(* CODESYS project DeanPowerSupplyComponent (1).library
   Author: Lily Dollard, Scott Kinder
   Version: 2025.10.20.11
   Title: Nemo
   Placeholder: Nemo
   Company: Photara

Project tree, tasks and I/O mapping:
  libraries: Base, 2025.10.13.11 (Photara); Tc2_Math, * (Beckhoff Automation GmbH); Tc2_Standard, * (Beckhoff Automation GmbH); Tc2_System, * (Beckhoff Automation GmbH); Tc2_Utilities, * (Beckhoff Automation GmbH)
  DUTs/
    data type ST_PowerSupplyCalibration
    data type ST_PowerSupplyConfiguration
    data type ST_PowerSupplyStatus
  GVLs/
    global variables GC_Dean
    global variables GPL_Dean
  ITFs/
    interface I_PowerSupply: Disable_HV, Enable_HV, InjectConfiguration, P_PowerSupplyStatus
    interface I_PowerSupplyConfiguration: P_PowerSupplyConfiguration
    interface I_PowerSupplyExt: GetCurrent, GetVoltage, InputPowerOff, InputPowerOn, SetCurrent, SetVoltage
    interface I_PowerSupplySystem: ClearErrors, Disable_HV, Enable_HV, FullShutDown, InputPowerOff, InputPowerOn, SetCurrent, SetVoltage
  POUs/
    function block FB_DeanPowerSupply [ST]: _DeanCyclic, _InitializeReferences, _SetCommandPermIntlkConfiguration, _UpdateComponentStatus, _ComponentCyclic, _EvaluateCompletionConditions, CyclicLogic, Disable_HV, Enable_HV, GetCurrent, GetVoltage, InputPowerOff, InputPowerOn, SetCurrent, SetVoltage, Check_Results, Test_Disable_HV, Test_Enable_HV, Test_GetCurrent, Test_GetVoltage, Test_InputPowerOff, Test_InputPowerOn, Test_SetCurrent, Test_SetVoltage, CheckForErrors, ClearErrors, InjectConfiguration, Interpolate, P_PowerSupplyConfiguration, P_PowerSupplyStatus
    function block FB_HVPS_System [ST]: _Initialize, _InitializeChildrenDependencies, _SetDependencyConfiguration, CyclicLogic, FB_Init, P_supply_status, RunTests, ClearErrors, Disable_HV, Enable_HV, FullShutDown, InputPowerOff, InputPowerOn, SetCurrent, SetVoltage
    program MAIN [ST]
  VISUs/
*)

// DUTs/ST_PowerSupplyCalibration
TYPE ST_PowerSupplyCalibration :
STRUCT
	VSET_Scale		: LREAL 	:= 1.000;
	VSET_Offset		: LREAL  := 0; // V
	ISET_Scale		: LREAL	:= 1.000;
	ISET_Offset		: LREAL  := 0; // mA
	                  
	VMON_Scale		: LREAL 	:= 1.000;
	VMON_Offset		: LREAL  := 0; // V
	IMON_Scale		: LREAL 	:= 1.000;
	IMON_Offset		: LREAL  := 0; // mA
END_STRUCT
END_TYPE

// DUTs/ST_PowerSupplyConfiguration
TYPE ST_PowerSupplyConfiguration :
STRUCT
	ComponentConfiguration : REFERENCE TO Base.ST_ComponentConfiguration;
	
	// Supply Characteristics
	IsPositive		: BOOL; 			// Sends negative monitor values to the HMI if False
	
	MinVoltage 		: LREAL := 0; 		// Minimum voltage (V) that the user can specify, usually 0
	MaxVoltageAbs 	: LREAL;			// Maximum voltage (V) that the user can specify
	MinCurrent		: LREAL := 0;		// Minimum current (mA) that the user can specify, usually 0
	MaxCurrent		: LREAL;			// Maximum current (mA) that the user can specify
	
	HasVMON			: BOOL 	:= TRUE; 	// Can the user watch the voltage output?
	HasIMON			: BOOL 	:= TRUE; 	// Can the user watch the current output?
	HasVSET			: BOOL 	:= TRUE;	// Can the user specify a desired voltage?
	HasISET			: BOOL 	:= TRUE; 	// Can the user specify maximum current?
	
	NeedsVREF		: BOOL ; 			// False if the reference voltage for control inputs is generated internally
	VREF			: LREAL;			// Reference voltage for control inputs
	plc_VREF		: INT;
	
	VSET_needs_ramp	: BOOL 	:= FALSE;	// False allows the full V value to be set immediately
	Ramp_increment	: LREAL := 10.0;   	// Voltage (V) to step up at a time after checking that current is within acceptable limits
	
	// Control signal characteristics
	plc_min_IMON  	: INT 	:= 0;    	// PLC signal corresponding to the minimum current reading
	plc_max_IMON  	: INT 	:= 32767; 	// PLC signal corresponding to the maximum current reading
	                                                                      
	plc_min_ISET  	: INT 	:= 0;	  	// PLC signal corresponding to the minimum current setting
	plc_max_ISET  	: INT 	:= 32767; 	// PLC signal corresponding to the maximum current setting
	
	plc_min_VMON  	: INT 	:= 0;     	// PLC signal corresponding to the minimum voltage reading
	plc_max_VMON  	: INT 	:= 32767;	// PLC signal corresponding to the maximum voltage reading
	                                                                         
	plc_min_VSET  	: INT 	:= 0;	  	// PLC signal corresponding to the minimum voltage setting
	plc_max_VSET  	: INT 	:= 32767; 	// PLC signal corresponding to the maximum voltage setting
	
	// Error Conditions
	OverCurrentErrorThreshold 		: LREAL := 1.05;	// over-current level, relative to IMON, to disable the output
	OverVoltageErrorThreshold 		: LREAL := 1.05;	// over-voltage level, relative to VSET, to disable the output
	MaxVoltageBuffer				: LREAL := 100.0;	// volts beyond MaxVoltageAbs to allow before killing supply power
	UnderVoltageWarningThreshold 	: LREAL := 0.95;	// under-voltage level, relative to VSET, to warn setpoint is not met
	
	ClearErrors : BOOL := FALSE;
	
	// Calibration
	Calibration		: ST_PowerSupplyCalibration;
	
	// Setpoints
	VSET			: LREAL;	// V
	ISET			: LREAL;	// mA
	POWERED			: BOOL;	
	ENABLED			: BOOL;
	
END_STRUCT
END_TYPE

// DUTs/ST_PowerSupplyStatus
TYPE ST_PowerSupplyStatus :
STRUCT
	BaseComponentStatus : REFERENCE TO Base.ST_ComponentStatus;
	
	// Controls mapped to PLC terminals
	VSET_to_plc 		AT %Q* : INT;
	ISET_to_plc 		AT %Q* : INT;
	VREF_to_plc			AT %Q* : INT;
	VMON_from_plc 		AT %I* : INT;
	IMON_from_plc 		AT %I* : INT;
	POWERED				AT %Q* : BOOL; 
	ENABLED				AT %Q* : BOOL;
	
	// Live outputs of the HV supply, translated into real units
	VMON 		: LREAL;	// V
	IMON		: LREAL;	// mA
	
	// Most recent settings given to the power supply
	VSET		: LREAL;
	ISET		: LREAL;
	
	V_was_set 	: BOOL; // flag for successful voltage set
	
	UnderVoltageWarning			: BOOL := FALSE;
	CurrentLimitWarning			: BOOL := FALSE;
	
	OverVoltageSetpointError	: BOOL := FALSE;
	OverMaxVoltageError			: BOOL := FALSE;
	
	OverCurrentSetpointError	: BOOL := FALSE;
	OverMaxCurrentError			: BOOL := FALSE;
	
	ErrorsAreClear					: BOOL := TRUE;
	
END_STRUCT
END_TYPE

// GVLs/GC_Dean
{attribute 'qualified_only'}
{attribute 'global_init_slot' := '41600'}
VAR_GLOBAL CONSTANT
	INDEX_COMMAND_MIN : DINT := GPL_Dean.INDEX_COMMAND_MIN;  
	INDEX_COMMAND_MAX : DINT := GPL_Dean.INDEX_COMMAND_MAX;
END_VAR

// GVLs/GPL_Dean
{attribute 'qualified_only'}
{attribute 'global_init_slot' := '41500'}
VAR_GLOBAL CONSTANT
	INDEX_COMMAND_MIN : DINT := 0;  
	INDEX_COMMAND_MAX : DINT := 5;
END_VAR

// ITFs/I_PowerSupply
// Basic high-voltage power supply that can turn on or off
INTERFACE I_PowerSupply EXTENDS I_BaseCyclic

// Shut off the output voltage
METHOD Disable_HV
VAR_INPUT
END_VAR
END_METHOD

// Turn on the output voltage
METHOD Enable_HV
VAR_INPUT
END_VAR
END_METHOD

METHOD InjectConfiguration
VAR_INPUT
	PowerSupplyConfiguration : REFERENCE TO ST_PowerSupplyConfiguration;
END_VAR
END_METHOD

PROPERTY P_PowerSupplyStatus : REFERENCE TO ST_PowerSupplyStatus
GET
END_GET
END_PROPERTY

END_INTERFACE

// ITFs/I_PowerSupplyConfiguration
// Basic high-voltage power supply that can turn on or off
INTERFACE I_PowerSupplyConfiguration EXTENDS __SYSTEM.IQueryInterface

PROPERTY P_PowerSupplyConfiguration : REFERENCE TO ST_PowerSupplyConfiguration
GET
END_GET
END_PROPERTY

END_INTERFACE

// ITFs/I_PowerSupplyExt
(*
Additional power supply capabilities:
* Adds a distinction between input power and the existing controls for HV output enable/disable
* Allows setting a desired output voltage and current
* Monitors the actual voltage and current
*)

INTERFACE I_PowerSupplyExt EXTENDS I_PowerSupply

// Read the currently-output current in milliamps (mA)
METHOD GetCurrent
END_METHOD

// Read the currently-output voltage in Volts (V)
METHOD GetVoltage
END_METHOD

// Turn off power to the supply
METHOD InputPowerOff
END_METHOD

// Turn on power to the supply
METHOD InputPowerOn
END_METHOD

// Send the the desired or maximum current setpoint (in mA) to the power supply
METHOD SetCurrent
VAR_INPUT
	setpoint : LREAL; // mA
END_VAR
END_METHOD

// Send the the voltage setpoint (V) to the power supply
METHOD SetVoltage
VAR_INPUT
	setpoint : LREAL; // V
END_VAR
END_METHOD

END_INTERFACE

// ITFs/I_PowerSupplySystem
INTERFACE I_PowerSupplySystem EXTENDS __SYSTEM.IQueryInterface

METHOD ClearErrors : BOOL
VAR_INPUT
	Index : DINT;
END_VAR
END_METHOD

(* Shut off the output voltage*)
METHOD Disable_HV
VAR_INPUT
	Index : DINT;
END_VAR
END_METHOD

{warning 'Add method implementation '}
(* Turn on the output voltage*)
METHOD Enable_HV
VAR_INPUT
	Index : DINT;
END_VAR
END_METHOD

METHOD FullShutDown : BOOL
VAR_INPUT
END_VAR
END_METHOD

{warning 'Add method implementation '}
(* Turn off power to the supply*)
METHOD InputPowerOff
VAR_INPUT
	Index : DINT;
END_VAR
END_METHOD

{warning 'Add method implementation '}
(* Turn on power to the supply*)
METHOD InputPowerOn
VAR_INPUT
	Index : DINT;
END_VAR
END_METHOD

{warning 'Add method implementation '}
(* Send the the desired or maximum current setpoint (in mA) to the power supply*)
METHOD SetCurrent
VAR_INPUT
	(* mA*)
	setpoint	: LREAL;
	Index : DINT;
END_VAR
END_METHOD

{warning 'Add method implementation '}
(* Send the the voltage setpoint (V) to the power supply*)
METHOD SetVoltage
VAR_INPUT
	(* V*)
	setpoint	: LREAL;
	Index : DINT;
END_VAR
END_METHOD

END_INTERFACE

// POUs/FB_DeanPowerSupply
FUNCTION_BLOCK FB_DeanPowerSupply EXTENDS Base.FB_Component<GC_Dean.INDEX_COMMAND_MIN,GC_Dean.INDEX_COMMAND_MAX> IMPLEMENTS I_PowerSupplyExt, I_PowerSupplyConfiguration
VAR CONSTANT
	INDEX_COMMAND_Enable_HV 		: INT := 0;
	INDEX_COMMAND_Disable_HV 		: INT := 1;
	INDEX_COMMAND_InputPowerOn		: INT := 2;
	INDEX_COMMAND_InputPowerOff 	: INT := 3;
	INDEX_COMMAND_SetVoltage 		: INT := 4;
	INDEX_COMMAND_SetCurrent		: INT := 5;
	
END_VAR

VAR
//	ComponentConfiguration : Base.ST_ComponentConfiguration;
	
//	_iInjectedConfiguration		: I_PowerSupplyConfiguration;
	
	Run_Tests_Trigger : BOOL := FALSE;
END_VAR

VAR_INPUT
	DeanConfig 		: ST_PowerSupplyConfiguration;
	DeanStatus		: ST_PowerSupplyStatus;
END_VAR

METHOD PROTECTED _DeanCyclic
VAR_INST
// 	VSET_actual	: LREAL;
// 	ISET_actual : LREAL;
END_VAR
// Reset errors if requested
IF DeanConfig.ClearErrors THEN
	ClearErrors();
	DeanConfig.ClearErrors := FALSE;
END_IF

// Turn on or off power if the config requests it
IF DeanStatus.POWERED <> DeanConfig.POWERED THEN
	IF DeanConfig.POWERED THEN
		InputPowerOn();
	ELSE
		InputPowerOff();
		DeanConfig.ENABLED := FALSE;
	END_IF
END_IF

// Enable or disable HV if the config requests it
IF DeanStatus.ENABLED <> DeanConfig.ENABLED THEN
	IF DeanConfig.ENABLED AND DeanConfig.POWERED THEN
		Enable_HV();
	ELSE
		DeanConfig.ENABLED := FALSE;
		Disable_HV();
	END_IF
END_IF

// get the actual last settings sent to the PLC (Config values are nominal)
// VSET_actual		:= DeanConfig.VSET * DeanConfig.Calibration.VSET_Scale + DeanConfig.Calibration.VSET_Offset;
// VSET_actual 	:= MAX(DeanConfig.MinVoltage, VSET_actual);
// VSET_actual 	:= MIN(VSET_actual, DeanConfig.MaxVoltageAbs);
// 
// ISET_actual		:= DeanConfig.ISET * DeanConfig.Calibration.ISET_Scale + DeanConfig.Calibration.ISET_Offset;
// ISET_actual 	:= MAX(DeanConfig.MinCurrent, ISET_actual);
// ISET_actual 	:= MIN(ISET_actual, DeanConfig.MaxCurrent);

// Send the desired values to the PLC if the input has changed
IF DeanConfig.HasVSET THEN
	// IF VSET_actual <> DeanStatus.VSET AND NOT (SUPER^.Commands[INDEX_COMMAND_SetVoltage].Busy) THEN
		SetVoltage(DeanConfig.VSET);
	// END_IF
END_IF

IF DeanConfig.HasISET THEN
	// IF ISET_actual <> DeanStatus.ISET THEN
		SetCurrent(DeanConfig.ISET);
	// END_IF
END_IF

// Monitor for errors (monitor pins only work when powered on)
IF DeanStatus.POWERED THEN
	CheckForErrors();
END_IF
END_METHOD

METHOD PROTECTED _InitializeReferences : BOOL
//Initialize data references
BaseConfiguration.InstancePath 						REF= InstancePath;

ComponentConfiguration.BaseConfiguration 			REF= SUPER^.BaseConfiguration;
                                                    
ComponentStatus.BaseStatus							REF= SUPER^.BaseStatus;

ComponentStatus.AmsNetId							REF= ComponentConfiguration.AmsNetId;

DeanConfig.ComponentConfiguration					REF= SUPER^.ComponentConfiguration;

DeanStatus.BaseComponentStatus						REF= SUPER^.ComponentStatus;

_InitializeReferences 								:= TRUE; // apply at end of all reference initialization
END_METHOD

METHOD PROTECTED _SetCommandPermIntlkConfiguration : BOOL
//Enable HV
CommandPermIntlkConfiguration[INDEX_COMMAND_Enable_HV].P_CommandConfiguration.CommandDescription := 'Enable Power Supply Output';
CommandPermIntlkConfiguration[INDEX_COMMAND_Enable_HV].P_CommandConfiguration.CommandIndex := INDEX_COMMAND_Enable_HV;
CommandPermIntlkConfiguration[INDEX_COMMAND_Enable_HV].P_CommandConfiguration.CommandPOUName := 'Enable_HV';
CommandPermIntlkConfiguration[INDEX_COMMAND_Enable_HV].P_CommandConfiguration.Priority := Base.E_CommandPriority.Priority_Normal;
CommandPermIntlkConfiguration[INDEX_COMMAND_Enable_HV].P_CommandConfiguration.TimeoutTime := T#200MS;
CommandPermIntlkConfiguration[INDEX_COMMAND_Enable_HV].P_CommandConfiguration.CompletionCondition REF= SUPER^.CommandCompletionConditions[INDEX_COMMAND_Enable_HV];

CommandPermIntlkConfiguration[INDEX_COMMAND_Enable_HV].P_PermIntlkConfiguration.PermIntlkObj[0].Condition REF= DeanStatus.POWERED;
CommandPermIntlkConfiguration[INDEX_COMMAND_Enable_HV].P_PermIntlkConfiguration.PermIntlkObj[0].Description := 'Powered on';
CommandPermIntlkConfiguration[INDEX_COMMAND_Enable_HV].P_PermIntlkConfiguration.PermIntlkObj[0].Index := 0;

CommandPermIntlkConfiguration[INDEX_COMMAND_Enable_HV].P_PermIntlkConfiguration.PermIntlkObj[1].Condition REF= DeanStatus.ErrorsAreClear;
CommandPermIntlkConfiguration[INDEX_COMMAND_Enable_HV].P_PermIntlkConfiguration.PermIntlkObj[1].Description := 'No voltage or current errors';
CommandPermIntlkConfiguration[INDEX_COMMAND_Enable_HV].P_PermIntlkConfiguration.PermIntlkObj[1].Index := 1;

//Disable HV
CommandPermIntlkConfiguration[INDEX_COMMAND_Disable_HV].P_CommandConfiguration.CommandDescription := 'Disable Power Supply Output';
CommandPermIntlkConfiguration[INDEX_COMMAND_Disable_HV].P_CommandConfiguration.CommandIndex := INDEX_COMMAND_Disable_HV;
CommandPermIntlkConfiguration[INDEX_COMMAND_Disable_HV].P_CommandConfiguration.CommandPOUName := 'Disable_HV';
CommandPermIntlkConfiguration[INDEX_COMMAND_Disable_HV].P_CommandConfiguration.Priority := Base.E_CommandPriority.Priority_High;
CommandPermIntlkConfiguration[INDEX_COMMAND_Disable_HV].P_CommandConfiguration.TimeoutTime := T#200MS;
CommandPermIntlkConfiguration[INDEX_COMMAND_Disable_HV].P_CommandConfiguration.CompletionCondition REF= SUPER^.CommandCompletionConditions[INDEX_COMMAND_Disable_HV];

//Input power on
CommandPermIntlkConfiguration[INDEX_COMMAND_InputPowerOn].P_CommandConfiguration.CommandDescription := 'Provide input power to supply';
CommandPermIntlkConfiguration[INDEX_COMMAND_InputPowerOn].P_CommandConfiguration.CommandIndex := INDEX_COMMAND_InputPowerOn;
CommandPermIntlkConfiguration[INDEX_COMMAND_InputPowerOn].P_CommandConfiguration.CommandPOUName := 'InputPowerOn';
CommandPermIntlkConfiguration[INDEX_COMMAND_InputPowerOn].P_CommandConfiguration.Priority := Base.E_CommandPriority.Priority_Normal;
CommandPermIntlkConfiguration[INDEX_COMMAND_InputPowerOn].P_CommandConfiguration.TimeoutTime := T#200MS;
CommandPermIntlkConfiguration[INDEX_COMMAND_InputPowerOn].P_CommandConfiguration.CompletionCondition REF= SUPER^.CommandCompletionConditions[INDEX_COMMAND_InputPowerOn];

CommandPermIntlkConfiguration[INDEX_COMMAND_InputPowerOn].P_PermIntlkConfiguration.PermIntlkObj[0].Condition REF= DeanStatus.ErrorsAreClear;
CommandPermIntlkConfiguration[INDEX_COMMAND_InputPowerOn].P_PermIntlkConfiguration.PermIntlkObj[0].Description := 'No voltage or current errors';
CommandPermIntlkConfiguration[INDEX_COMMAND_InputPowerOn].P_PermIntlkConfiguration.PermIntlkObj[0].Index := 0;

//Input power off
CommandPermIntlkConfiguration[INDEX_COMMAND_InputPowerOff].P_CommandConfiguration.CommandDescription := 'Cut off input power to supply';
CommandPermIntlkConfiguration[INDEX_COMMAND_InputPowerOff].P_CommandConfiguration.CommandIndex := INDEX_COMMAND_InputPowerOff;
CommandPermIntlkConfiguration[INDEX_COMMAND_InputPowerOff].P_CommandConfiguration.CommandPOUName := 'InputPowerOff';
CommandPermIntlkConfiguration[INDEX_COMMAND_InputPowerOff].P_CommandConfiguration.Priority := Base.E_CommandPriority.Priority_High;
CommandPermIntlkConfiguration[INDEX_COMMAND_InputPowerOff].P_CommandConfiguration.TimeoutTime := T#200MS;
CommandPermIntlkConfiguration[INDEX_COMMAND_InputPowerOff].P_CommandConfiguration.CompletionCondition REF= SUPER^.CommandCompletionConditions[INDEX_COMMAND_InputPowerOff];

//Set Voltage
CommandPermIntlkConfiguration[INDEX_COMMAND_SetVoltage].P_CommandConfiguration.CommandDescription := 'Set the desired HV output voltage';
CommandPermIntlkConfiguration[INDEX_COMMAND_SetVoltage].P_CommandConfiguration.CommandIndex := INDEX_COMMAND_SetVoltage;
CommandPermIntlkConfiguration[INDEX_COMMAND_SetVoltage].P_CommandConfiguration.CommandPOUName := 'SetVoltage';
CommandPermIntlkConfiguration[INDEX_COMMAND_SetVoltage].P_CommandConfiguration.Priority := Base.E_CommandPriority.Priority_Normal;
CommandPermIntlkConfiguration[INDEX_COMMAND_SetVoltage].P_CommandConfiguration.TimeoutTime := T#200MS;
CommandPermIntlkConfiguration[INDEX_COMMAND_SetVoltage].P_CommandConfiguration.CompletionCondition REF= SUPER^.CommandCompletionConditions[INDEX_COMMAND_SetVoltage];

CommandPermIntlkConfiguration[INDEX_COMMAND_SetVoltage].P_PermIntlkConfiguration.PermIntlkObj[0].Condition REF= DeanConfig.HasVSET;
CommandPermIntlkConfiguration[INDEX_COMMAND_SetVoltage].P_PermIntlkConfiguration.PermIntlkObj[0].Description := 'HVPS has VSET capability';
CommandPermIntlkConfiguration[INDEX_COMMAND_SetVoltage].P_PermIntlkConfiguration.PermIntlkObj[0].Index := 0;

CommandPermIntlkConfiguration[INDEX_COMMAND_SetVoltage].P_PermIntlkConfiguration.PermIntlkObj[1].Condition REF= DeanStatus.POWERED;
CommandPermIntlkConfiguration[INDEX_COMMAND_SetVoltage].P_PermIntlkConfiguration.PermIntlkObj[1].Description := 'Supply power is on, can set voltage';
CommandPermIntlkConfiguration[INDEX_COMMAND_SetVoltage].P_PermIntlkConfiguration.PermIntlkObj[1].Index := 1;

//Set Current
CommandPermIntlkConfiguration[INDEX_COMMAND_SetCurrent].P_CommandConfiguration.CommandDescription := 'Set the maximum current output from the HV terminals';
CommandPermIntlkConfiguration[INDEX_COMMAND_SetCurrent].P_CommandConfiguration.CommandIndex := INDEX_COMMAND_SetCurrent;
CommandPermIntlkConfiguration[INDEX_COMMAND_SetCurrent].P_CommandConfiguration.CommandPOUName := 'SetCurrent';
CommandPermIntlkConfiguration[INDEX_COMMAND_SetCurrent].P_CommandConfiguration.Priority := Base.E_CommandPriority.Priority_Normal;
CommandPermIntlkConfiguration[INDEX_COMMAND_SetCurrent].P_CommandConfiguration.TimeoutTime := T#200MS;
CommandPermIntlkConfiguration[INDEX_COMMAND_SetCurrent].P_CommandConfiguration.CompletionCondition REF= SUPER^.CommandCompletionConditions[INDEX_COMMAND_SetCurrent];

CommandPermIntlkConfiguration[INDEX_COMMAND_SetCurrent].P_PermIntlkConfiguration.PermIntlkObj[0].Condition REF= DeanConfig.HasISET;
CommandPermIntlkConfiguration[INDEX_COMMAND_SetCurrent].P_PermIntlkConfiguration.PermIntlkObj[0].Description := 'HVPS has ISET capability';
CommandPermIntlkConfiguration[INDEX_COMMAND_SetCurrent].P_PermIntlkConfiguration.PermIntlkObj[0].Index := 0;

CommandPermIntlkConfiguration[INDEX_COMMAND_SetCurrent].P_PermIntlkConfiguration.PermIntlkObj[1].Condition REF= DeanStatus.POWERED;
CommandPermIntlkConfiguration[INDEX_COMMAND_SetCurrent].P_PermIntlkConfiguration.PermIntlkObj[1].Description := 'Supply power is on, can set current';
CommandPermIntlkConfiguration[INDEX_COMMAND_SetCurrent].P_PermIntlkConfiguration.PermIntlkObj[1].Index := 1;

_SetCommandPermIntlkConfiguration := TRUE;
END_METHOD

METHOD PROTECTED _UpdateComponentStatus : Base.I_ComponentFull
// Update the parts of status that need to be monitored continuously
IF DeanConfig.POWERED THEN
	IF DeanConfig.HasVMON THEN
		GetVoltage();
	END_IF
	IF DeanConfig.HasIMON THEN
		GetCurrent();
	END_IF
END_IF

_UpdateComponentStatus := THIS^;
END_METHOD

METHOD PROTECTED _ComponentCyclic : Base.I_ComponentFull
_ComponentCyclic := THIS^;
END_METHOD

(*
Example Implementation:
// Set completion conditions - commands complete immediately after transitioning to acting state
// This prevents the component from staying busy and blocking other commands
SUPER^.CommandCompletionConditions[INDEX_COMMAND_ABORT]            		:= (SequencerStatus.CurrentState = E_PackMLState.Aborting);
SUPER^.CommandCompletionConditions[INDEX_COMMAND_CLEAR]            		:= (SequencerStatus.CurrentState = E_PackMLState.Clearing);
SUPER^.CommandCompletionConditions[INDEX_COMMAND_COMPLETE]         		:= (SequencerStatus.CurrentState = E_PackMLState.Completing);
SUPER^.CommandCompletionConditions[INDEX_COMMAND_HOLD]             		:= (SequencerStatus.CurrentState = E_PackMLState.Holding);
SUPER^.CommandCompletionConditions[INDEX_COMMAND_RESET]            		:= (SequencerStatus.CurrentState = E_PackMLState.Resetting);
SUPER^.CommandCompletionConditions[INDEX_COMMAND_RESUMEFROMHOLD]   		:= (SequencerStatus.CurrentState = E_PackMLState.Unholding);
SUPER^.CommandCompletionConditions[INDEX_COMMAND_RESUMEFROMSUSPEND]		:= (SequencerStatus.CurrentState = E_PackMLState.Unsuspending);
SUPER^.CommandCompletionConditions[INDEX_COMMAND_START]            		:= (SequencerStatus.CurrentState = E_PackMLState.Starting);
SUPER^.CommandCompletionConditions[INDEX_COMMAND_STOP]             		:= (SequencerStatus.CurrentState = E_PackMLState.Stopping);
SUPER^.CommandCompletionConditions[INDEX_COMMAND_SUSPEND]          		:= (SequencerStatus.CurrentState = E_PackMLState.Suspending);

// Enable/Disable don't have specific PackML states, handle as needed
SUPER^.CommandCompletionConditions[INDEX_COMMAND_ENABLE]           		:= (NOT SUPER^.BaseStatus.Enabled);
SUPER^.CommandCompletionConditions[INDEX_COMMAND_DISABLE]          		:= SUPER^.BaseStatus.Enabled;

_EvaluateCompletionConditions	:= TRUE;
*)
METHOD PROTECTED _EvaluateCompletionConditions : BOOL
// Set completion conditions - commands complete immediately after transitioning to acting state
// This prevents the component from staying busy and blocking other commands
SUPER^.CommandCompletionConditions[INDEX_COMMAND_Enable_HV]            	:= DeanStatus.ENABLED;
SUPER^.CommandCompletionConditions[INDEX_COMMAND_Disable_HV]            := NOT(DeanStatus.ENABLED);
SUPER^.CommandCompletionConditions[INDEX_COMMAND_InputPowerOn]          := DeanStatus.POWERED;
SUPER^.CommandCompletionConditions[INDEX_COMMAND_InputPowerOff]         := NOT(DeanStatus.POWERED);
SUPER^.CommandCompletionConditions[INDEX_COMMAND_SetVoltage]            := DeanStatus.V_was_set;
SUPER^.CommandCompletionConditions[INDEX_COMMAND_SetCurrent]            := DeanStatus.ISET = DeanConfig.ISET;

_EvaluateCompletionConditions	:= TRUE;
END_METHOD

METHOD CyclicLogic
SUPER^.CyclicLogic();

_ComponentCyclic();

_DeanCyclic();
END_METHOD

METHOD Disable_HV
VAR_INPUT
END_VAR
// ExecuteCommand(CmdIndex := INDEX_COMMAND_Disable_HV);

// IF SUPER^.iCommands[INDEX_COMMAND_Disable_HV].P_CommandStatus.Result = E_CommandResult.Accepted THEN
	DeanStatus.ENABLED := FALSE;
// END_IF
END_METHOD

METHOD Enable_HV
VAR_INPUT
END_VAR
// ExecuteCommand(CmdIndex := INDEX_COMMAND_Enable_HV);

// IF SUPER^.iCommands[INDEX_COMMAND_Enable_HV].P_CommandStatus.Result = E_CommandResult.Accepted THEN
	DeanStatus.ENABLED := TRUE;
// END_IF
END_METHOD

(* Read the currently-output current in milliamps (mA)*)
METHOD GetCurrent
VAR
	raw_current			: LREAL;	// mA
	calibrated_current	: LREAL;	// mA
END_VAR
IF DeanConfig.HasIMON THEN
	raw_current := ABS( Interpolate( Input		:= DeanStatus.IMON_from_plc,
									 Input_min	:= DeanConfig.plc_min_IMON,
									 Input_max	:= DeanConfig.plc_max_IMON,
									 Output_min	:= DeanConfig.MinCurrent,
									 Output_max	:= DeanConfig.MaxCurrent));
	
	calibrated_current := raw_current * DeanConfig.Calibration.IMON_Scale + DeanConfig.Calibration.IMON_Offset;
	DeanStatus.IMON := calibrated_current;
END_IF
END_METHOD

(* Read the currently-output voltage in Volts (V)*)
METHOD GetVoltage
VAR
	raw_HV			: LREAL;	// V
	calibrated_HV	: LREAL;	// V
END_VAR
IF DeanConfig.HasVMON THEN
	raw_HV := ABS( Interpolate( Input		:= DeanStatus.VMON_from_plc,
								Input_min	:= DeanConfig.plc_min_VMON,
								Input_max	:= DeanConfig.plc_max_VMON,
								Output_min	:= DeanConfig.MinVoltage,
								Output_max	:= DeanConfig.MaxVoltageAbs));
	
	calibrated_HV := raw_HV * DeanConfig.Calibration.VMON_Scale + DeanConfig.Calibration.VMON_Offset;
	DeanStatus.VMON := calibrated_HV;
END_IF
END_METHOD

(* Turn off power to the supply *)
METHOD InputPowerOff
// ExecuteCommand(CmdIndex := INDEX_COMMAND_InputPowerOff);

// IF SUPER^.iCommands[INDEX_COMMAND_InputPowerOff].P_CommandStatus.Result = E_CommandResult.Accepted THEN
	DeanStatus.POWERED := FALSE;
	IF DeanConfig.NeedsVREF THEN
		DeanStatus.VREF_to_plc := 0;
	END_IF
// END_IF
END_METHOD

(* Turn off power to the supply *)
METHOD InputPowerOn
// ExecuteCommand(CmdIndex := INDEX_COMMAND_InputPowerOn);

// IF SUPER^.iCommands[INDEX_COMMAND_InputPowerOn].P_CommandStatus.Result = E_CommandResult.Accepted THEN
	DeanStatus.POWERED := TRUE;
	IF DeanConfig.NeedsVREF THEN
		DeanStatus.VREF_to_plc := DeanConfig.plc_VREF;
	END_IF
// END_IF
END_METHOD

(* Send the the desired or maximum current setpoint (in mA) to the power supply*)
METHOD SetCurrent
VAR_INPUT
	setpoint : LREAL; // mA
END_VAR
VAR
	setpoint_adjusted 	: LREAL; // mA
	output				: INT;
END_VAR
// ExecuteCommand(CmdIndex := INDEX_COMMAND_SetCurrent);

// IF SUPER^.iCommands[INDEX_COMMAND_SetCurrent].P_CommandStatus.Result = E_CommandResult.Accepted THEN
	// Convert to positive for all internal calculations
	setpoint_adjusted := ABS(setpoint);
	// Apply calibration
	setpoint_adjusted := setpoint_adjusted * DeanConfig.Calibration.ISET_Scale +  DeanConfig.Calibration.ISET_Offset;
	// Apply current restrictions
	setpoint_adjusted := MAX(DeanConfig.MinCurrent, setpoint_adjusted);
	setpoint_adjusted := MIN(setpoint_adjusted, DeanConfig.MaxCurrent);
	
	// Project setpoint onto the terminal range
	output :=  LREAL_TO_INT( Interpolate(	Input      := setpoint_adjusted,
											Input_min  := DeanConfig.MinCurrent,
											Input_max  := DeanConfig.MaxCurrent,
											Output_min := DeanConfig.plc_min_ISET,
											Output_max := DeanConfig.plc_max_ISET ));
	// Send output to the terminal									 
	DeanStatus.ISET_to_plc := output;
	
	// Update the ISET status with the last confirmed setpoint
	DeanStatus.ISET := setpoint_adjusted;
// END_IF
END_METHOD

(* Send the the voltage setpoint (V) to the power supply*)
METHOD SetVoltage
VAR_INPUT
	setpoint : LREAL; // V
END_VAR
VAR
	setpoint_adjusted 	: LREAL; // V
	output				: INT;
END_VAR
DeanStatus.V_was_set := FALSE;

// ExecuteCommand(CmdIndex := INDEX_COMMAND_SetVoltage);

// IF SUPER^.iCommands[INDEX_COMMAND_SetVoltage].P_CommandStatus.Result = E_CommandResult.Accepted THEN
	// Convert to positive for all internal calculations
	setpoint_adjusted := ABS(setpoint);
	// Apply calibration
	setpoint_adjusted := setpoint_adjusted * DeanConfig.Calibration.VSET_Scale +  DeanConfig.Calibration.VSET_Offset;
	
	// Ramping behavior (requires IMON)
	IF DeanConfig.VSET_needs_ramp AND DeanConfig.HasIMON AND setpoint_adjusted > DeanStatus.VSET THEN 							// If ramping is required and possible, and the voltage is increasing // TODO add a check in the init that forbids requiring a ramp without an IMON
		IF 	(DeanConfig.HasISET AND DeanStatus.IMON <= DeanConfig.ISET)
		 OR ((NOT DeanConfig.HasISET) AND DeanStatus.IMON <= DeanConfig.MaxCurrent) THEN 											// if current is below nominal limit
			setpoint_adjusted := MIN(setpoint_adjusted, DeanStatus.VSET + DeanConfig.Ramp_increment); 									// make the setpoint higher than the last setpoint by the increment
		ELSE 																														// else (current too high)
			setpoint_adjusted := DeanStatus.VSET; 																						// leave the setpoint the same as the previous setpoint
		END_IF
	END_IF
	
	// Apply voltage restrictions
	setpoint_adjusted := MAX(DeanConfig.MinVoltage, setpoint_adjusted);
	setpoint_adjusted := MIN(setpoint_adjusted, DeanConfig.MaxVoltageAbs);
	
	// Project setpoint onto the terminal range
	output :=  LREAL_TO_INT( Interpolate(	Input      := setpoint_adjusted,
											Input_min  := DeanConfig.MinVoltage,
											Input_max  := DeanConfig.MaxVoltageAbs,
											Output_min := DeanConfig.plc_min_VSET,
											Output_max := DeanConfig.plc_max_VSET ));
	// Send output to the terminal									 
	DeanStatus.VSET_to_plc := output;
	
	// Update the VSET status with the last confirmed setpoint
	DeanStatus.VSET := setpoint_adjusted;
	
	// Confirm operation ran successfully
	DeanStatus.V_was_set := TRUE;
	
// END_IF
END_METHOD

METHOD Check_Results : BOOL
VAR_IN_OUT
	results : ARRAY[*] OF BOOL;
END_VAR
VAR_INPUT
	test_name : T_MaxString;
	log_summary : BOOL := TRUE;
END_VAR
VAR
	loop_index 		: DINT := 0;
	tests_passed 	: INT := 0;
	loop_index_string 	: T_MaxString;
	summary_string		: T_MaxString := CONCAT(test_name, ' tests passed: ');
	fail_string			: T_MaxString := CONCAT(test_name, ' test failed: ');
END_VAR
FOR loop_index := LOWER_BOUND(results, 1) TO UPPER_BOUND(results, 1) DO
	loop_index_string := TO_STRING(TO_INT(loop_index) + 1);
	IF results[loop_index] THEN
		tests_passed := tests_passed + 1;
	ELSE
		TraceWithSeverity(Message := CONCAT(fail_string, loop_index_string), Severity := Global.TcEventSeverity.Error); // TODO: Say the name of the test instead of the index
	END_IF
END_FOR

summary_string := CONCAT(summary_string, TO_STRING(tests_passed));
summary_string := CONCAT(summary_string, '/');
summary_string := CONCAT(summary_string, loop_index_string);
IF log_summary THEN
	TraceWithSeverity(Message := summary_string, Severity := Global.TcEventSeverity.Error);
END_IF

IF tests_passed = loop_index THEN
	Check_Results := TRUE;
ELSE
	Check_Results := FALSE;
END_IF
END_METHOD

METHOD Test_Disable_HV : BOOL
VAR_INPUT
END_VAR
VAR CONSTANT
	num_tests : INT := 1;
	POU_Name : T_MaxString := 'Disable_HV()';
END_VAR
VAR
	results : ARRAY [0..num_tests - 1] OF BOOL; // Initializes to false (failed test)
	test_index : INT;
END_VAR
// Test cases for the method Disable_HV()

// Test 1: Attempt to disable
test_index := 0;

DeanStatus.ENABLED := TRUE;
Disable_HV();

IF NOT(DeanStatus.ENABLED) THEN
	results[test_index] := TRUE;
END_IF

// Reset state
DeanStatus.ENABLED := FALSE;
DeanStatus.POWERED := FALSE;

// Check and return results
Test_Disable_HV := Check_Results(results, POU_Name, log_summary := FALSE);
END_METHOD

METHOD Test_Enable_HV : BOOL
VAR_INPUT
END_VAR
VAR CONSTANT
	num_tests : INT := 3;
	POU_Name : T_MaxString := 'Enable_HV()';
END_VAR
VAR
	results : ARRAY [0..num_tests - 1] OF BOOL; // Initializes to false (failed test)
	test_index : INT;
END_VAR
// Test cases for the method Enable_HV()

// Test 1: Attempt to enable while powered off (forbidden)
test_index := 0;

DeanStatus.ENABLED		:= FALSE;
DeanStatus.POWERED 		:= FALSE;
DeanStatus.ErrorsAreClear 	:= TRUE;

Enable_HV();

IF NOT(DeanStatus.ENABLED) THEN
	results[test_index] := TRUE;
END_IF


// Test 2: Attempt to enable while powered on (allowed)
test_index := test_index + 1;

DeanStatus.ENABLED		:= FALSE;
DeanStatus.POWERED 		:= TRUE;
DeanStatus.ErrorsAreClear 	:= TRUE;

Enable_HV();

IF DeanStatus.ENABLED THEN
	results[test_index] := TRUE;
END_IF

// Test 3: Attempt to enable during error state (forbidden)
test_index := test_index + 1;

DeanStatus.ENABLED		:= FALSE;
DeanStatus.POWERED 		:= TRUE;
DeanStatus.ErrorsAreClear 	:= FALSE;

Enable_HV();

IF NOT(DeanStatus.ENABLED) THEN
	results[test_index] := TRUE;
END_IF


// Reset state
DeanStatus.ENABLED := FALSE;
DeanStatus.POWERED := FALSE;

// Check and return results
Test_Enable_HV := Check_Results(results, POU_Name, log_summary := FALSE);
END_METHOD

METHOD Test_GetCurrent : BOOL
VAR_INPUT
END_VAR
VAR CONSTANT
	num_tests : INT := 2;
	POU_Name : T_MaxString := 'GetCurrent()';
END_VAR
VAR
	results : ARRAY [0..num_tests - 1] OF BOOL; // Initializes to false (failed test)
	test_index : INT;
END_VAR
// Test cases for the method GetCurrent()

// TODO: Attempt to handle erroneous inputs
// TODO: Check that calibration is working

// These tests assume base calibration and open permissives for now
DeanConfig.Calibration.IMON_Scale  := 1.0;
DeanConfig.Calibration.IMON_Offset := 0.0;

DeanStatus.POWERED 		:= TRUE;
DeanStatus.ENABLED 		:= TRUE;
DeanConfig.HasIMON 		:= TRUE;

// Test 1: Attempt to get current when reading is 0
test_index := 0;

DeanStatus.IMON_from_plc := 0;
DeanStatus.IMON := 2.0; // non zero to start

GetCurrent();

IF DeanStatus.IMON = 0.0 THEN
	results[test_index] := TRUE;
END_IF

// Test 2: Attempt to get current when reading at the maximum
test_index := test_index + 1;

DeanStatus.IMON := 0.0;
DeanStatus.IMON_from_plc := DeanConfig.plc_max_IMON;

GetCurrent();

IF DeanStatus.IMON = DeanConfig.MaxCurrent THEN
	results[test_index] := TRUE;
END_IF


// Check and return results
Test_GetCurrent := Check_Results(results, POU_Name, log_summary := FALSE);
END_METHOD

METHOD Test_GetVoltage : BOOL
VAR_INPUT
END_VAR
VAR CONSTANT
	num_tests : INT := 2;
	POU_Name : T_MaxString := 'GetVoltage()';
END_VAR
VAR
	results : ARRAY [0..num_tests - 1] OF BOOL; // Initializes to false (failed test)
	test_index : INT;
END_VAR
// Test cases for the method GetVoltage()

// TODO: Attempt to handle erroneous inputs
// TODO: Check that calibration is working

// These tests assume base calibration and open permissives for now
DeanConfig.Calibration.VMON_Scale  := 1.0;
DeanConfig.Calibration.VMON_Offset := 0.0;

DeanStatus.POWERED 		:= TRUE;
DeanStatus.ENABLED 		:= TRUE;
DeanConfig.HasVMON 		:= TRUE;

// Test 1: Attempt to get voltage when reading is 0
test_index := 0;

DeanStatus.VMON_from_plc := 0;
DeanStatus.VMON := 2.0; // non zero to start

GetVoltage();

IF DeanStatus.VMON = 0.0 THEN
	results[test_index] := TRUE;
END_IF

// Test 2: Attempt to get voltage when reading at the maximum
test_index := test_index + 1;

DeanStatus.VMON := 0.0;
DeanStatus.VMON_from_plc := DeanConfig.plc_max_VMON;

GetVoltage();

IF DeanStatus.VMON = DeanConfig.MaxVoltageAbs THEN
	results[test_index] := TRUE;
END_IF


// Check and return results
Test_GetVoltage := Check_Results(results, POU_Name, log_summary := FALSE);
END_METHOD

METHOD Test_InputPowerOff : BOOL
VAR_INPUT
END_VAR
VAR CONSTANT
	num_tests : INT := 1;
	POU_Name : T_MaxString := 'InputPowerOff()';
END_VAR
VAR
	results : ARRAY [0..num_tests - 1] OF BOOL; // Initializes to false (failed test)
	test_index : INT;
END_VAR
// Test cases for the method InputPowerOn()

// Test 1: Attempt to power off (always allowed)
test_index := 0;

DeanStatus.POWERED := TRUE;
InputPowerOff();

IF NOT(DeanStatus.POWERED) THEN
	results[test_index] := TRUE;
END_IF

// Reset state
DeanStatus.POWERED := FALSE;

// Check and return results
Test_InputPowerOff := Check_Results(results, POU_Name, log_summary := FALSE);
END_METHOD

METHOD Test_InputPowerOn : BOOL
VAR_INPUT
END_VAR
VAR CONSTANT
	num_tests : INT := 2;
	POU_Name : T_MaxString := 'InputPowerOn()';
END_VAR
VAR
	results : ARRAY [0..num_tests - 1] OF BOOL; // Initializes to false (failed test)
	test_index : INT;
END_VAR
// Test cases for the method InputPowerOn()

// Test 1: Attempt to power on under normal conditions (allowed)
test_index := 0;

DeanStatus.POWERED 		:= FALSE;
DeanStatus.ErrorsAreClear	:= TRUE;
InputPowerOn();

IF DeanStatus.POWERED THEN
	results[test_index] := TRUE;
END_IF

// Test 2: Attempt to power on during error state (forbidden)
test_index := test_index + 1;

DeanStatus.POWERED	 	:= FALSE;
DeanStatus.ErrorsAreClear 	:= FALSE;
InputPowerOn();

IF NOT(DeanStatus.POWERED) THEN
	results[test_index] := TRUE;
END_IF

// Reset state
DeanStatus.POWERED := FALSE;

// Check and return results
Test_InputPowerOn := Check_Results(results, POU_Name, log_summary := FALSE);
END_METHOD

METHOD Test_SetCurrent : BOOL
VAR_INPUT
END_VAR
VAR CONSTANT
	num_tests : INT := 3;
	POU_Name : T_MaxString := 'SetCurrent()';
END_VAR
VAR
	results : ARRAY [0..num_tests - 1] OF BOOL; // Initializes to false (failed test)
	test_index : INT;
END_VAR
// Test cases for the method SetCurrent()

// TODO: Attempt to thwart nefarious inputs
// TODO: Check that calibration is working

// These tests assume base calibration for now
DeanConfig.Calibration.ISET_Scale  := 1.0;
DeanConfig.Calibration.ISET_Offset := 0.0;
DeanConfig.HasISET := TRUE;

// Test 1: Attempt to set current while powered off (forbidden)
test_index := 0;

DeanStatus.ENABLED 		:= FALSE;
DeanStatus.POWERED 		:= FALSE;
DeanStatus.ISET			:= DeanConfig.MinCurrent;
DeanStatus.ISET_to_plc 	:= DeanConfig.plc_min_ISET;

SetCurrent(0.3);

IF DeanStatus.ISET = 0 AND DeanStatus.ISET_to_plc = DeanConfig.plc_min_ISET THEN
	results[test_index] := TRUE;
END_IF


// Test 2: Attempt to set current to max while powered on (allowed)
test_index := test_index + 1;

DeanStatus.ENABLED 		:= TRUE;
DeanStatus.POWERED 		:= TRUE;
DeanStatus.ISET			:= DeanConfig.MinCurrent;
DeanStatus.ISET_to_plc 	:= DeanConfig.plc_min_ISET;

SetCurrent(DeanConfig.MaxCurrent);

IF DeanStatus.ISET = DeanConfig.MaxCurrent AND DeanStatus.ISET_to_plc = DeanConfig.plc_max_ISET THEN
	results[test_index] := TRUE;
END_IF

// Test 2: Attempt to set current to 0 while powered on (allowed)
test_index := test_index + 1;

DeanStatus.ENABLED 		:= TRUE;
DeanStatus.POWERED 		:= TRUE;
DeanStatus.ISET			:= DeanConfig.MaxCurrent;
DeanStatus.ISET_to_plc 	:= DeanConfig.plc_max_ISET;
SetCurrent(DeanConfig.MinCurrent);

IF DeanStatus.ISET = DeanConfig.MinCurrent AND DeanStatus.ISET_to_plc = DeanConfig.plc_min_ISET THEN
	results[test_index] := TRUE;
END_IF

// Reset state
DeanStatus.ENABLED 		:= FALSE;
DeanStatus.POWERED 		:= FALSE;
DeanStatus.ISET			:= DeanConfig.MinCurrent;
DeanStatus.ISET_to_plc 	:= DeanConfig.plc_min_ISET;

// Check and return results
Test_SetCurrent := Check_Results(results, POU_Name, log_summary := FALSE);
END_METHOD

METHOD Test_SetVoltage : BOOL
VAR_INPUT
END_VAR
VAR CONSTANT
	num_tests : INT := 4;
	POU_Name : T_MaxString := 'SetVoltage()';
END_VAR
VAR
	results : ARRAY [0..num_tests - 1] OF BOOL; // Initializes to false (failed test)
	test_index : INT;
END_VAR
// Test cases for the method SetVoltage()

// TODO: Attempt to thwart nefarious inputs
// TODO: Check that calibration is working

// These tests assume base calibration for now
DeanConfig.Calibration.VSET_Scale  := 1.0;
DeanConfig.Calibration.VSET_Offset := 0.0;
DeanConfig.HasVSET := TRUE;

// Test 1: Attempt to set voltage while powered off (forbidden)
test_index := 0;

DeanStatus.ENABLED 		:= FALSE;
DeanStatus.POWERED 		:= FALSE;
DeanStatus.VSET			:= DeanConfig.MinVoltage;
DeanStatus.VSET_to_plc 	:= DeanConfig.plc_min_VSET;
SetVoltage(500);

IF DeanStatus.VSET = 0 AND DeanStatus.VSET_to_plc = DeanConfig.plc_min_VSET THEN
	results[test_index] := TRUE;
END_IF

// Test 2: Attempt to set voltage to 0 while powered on (allowed)
test_index := test_index + 1;

DeanStatus.ENABLED 		:= TRUE;
DeanStatus.POWERED 		:= TRUE;
DeanStatus.VSET			:= DeanConfig.MaxCurrent;
DeanStatus.VSET_to_plc 	:= DeanConfig.plc_max_VSET;

SetVoltage(DeanConfig.MinCurrent);

IF DeanStatus.VSET = DeanConfig.MinVoltage AND DeanStatus.VSET_to_plc = DeanConfig.plc_min_VSET THEN
	results[test_index] := TRUE;
END_IF

// Test 3: Attempt to set voltage to max while powered on, no ramp(allowed, should set instantly)
test_index := test_index + 1;

DeanStatus.ENABLED 		:= TRUE;
DeanStatus.POWERED 		:= TRUE;
DeanStatus.VSET			:= DeanConfig.MinVoltage;
DeanStatus.VSET_to_plc 	:= DeanConfig.plc_min_VSET;
DeanConfig.VSET_needs_ramp	:= FALSE;

SetVoltage(DeanConfig.MaxVoltageAbs);

IF DeanStatus.VSET = DeanConfig.MaxVoltageAbs AND DeanStatus.VSET_to_plc = DeanConfig.plc_max_VSET THEN
	results[test_index] := TRUE;
END_IF

// Test 4: Attempt to set voltage to max while powered on, ramp (allowed, should increase only by ramp amount)
test_index := test_index + 1;

DeanStatus.ENABLED 			:= TRUE;
DeanStatus.POWERED 			:= TRUE;
DeanStatus.VSET				:= DeanConfig.MinVoltage;
DeanStatus.VSET_to_plc 		:= DeanConfig.plc_min_VSET;
DeanConfig.VSET_needs_ramp		:= TRUE;
DeanConfig.Ramp_increment 	:= 30;
DeanStatus.IMON				:= 0.0;

SetVoltage(DeanConfig.MaxVoltageAbs);

IF DeanStatus.VSET = DeanConfig.MinVoltage + DeanConfig.Ramp_increment THEN
	results[test_index] := TRUE;
END_IF

// Reset state
DeanStatus.ENABLED 		:= FALSE;
DeanStatus.POWERED 		:= FALSE;
DeanStatus.VSET			:= DeanConfig.MinCurrent;
DeanStatus.VSET_to_plc 	:= DeanConfig.plc_min_VSET;

// Check and return results
Test_SetVoltage := Check_Results(results, POU_Name, log_summary := FALSE);
END_METHOD

METHOD CheckForErrors : BOOL
VAR_INPUT
END_VAR
ClearErrors();
RETURN;

// Check for warnings and reset warning flags if conditions are OK
IF 		DeanConfig.HasIMON
	AND DeanConfig.HasISET
	AND DeanStatus.IMON >= DeanConfig.ISET
	AND DeanConfig.ISET > 0
	AND NOT(DeanStatus.CurrentLimitWarning) THEN
	
	TraceWithSeverity(Message := 'Current limit reached', severity := TcEventSeverity.Warning);
	DeanStatus.CurrentLimitWarning := TRUE;
ELSE
	DeanStatus.CurrentLimitWarning := FALSE;
END_IF

IF		DeanConfig.HasVMON
	AND DeanConfig.HasVSET
	AND DeanStatus.VMON <= DeanConfig.VSET * DeanConfig.UnderVoltageWarningThreshold
	AND DeanConfig.VSET > 0
	AND NOT(DeanStatus.UnderVoltageWarning) THEN
	
	TraceWithSeverity(Message := 'Voltage below setpoint', severity := TcEventSeverity.Warning);
	DeanStatus.UnderVoltageWarning := TRUE;
ELSE
	DeanStatus.UnderVoltageWarning := FALSE;
END_IF


// Check for errors, do not reset if conditions are OK - resetting requires a call to ClearErrors()
IF 		DeanConfig.HasIMON
	AND DeanStatus.IMON > DeanConfig.MaxCurrent 
	THEN
	
	Disable_HV();
	InputPowerOff();
	
	IF NOT(DeanStatus.OverMaxCurrentError) THEN
		DeanStatus.OverMaxCurrentError := TRUE;
		TraceWithSeverity(Message := 'HVPS max output current exceeded', severity := TcEventSeverity.Critical);
	END_IF
	
ELSIF 	DeanConfig.HasISET
	AND DeanConfig.HasIMON
	AND DeanStatus.IMON > (DeanConfig.OverCurrentErrorThreshold * DeanConfig.ISET)
	AND DeanConfig.ISET > 0 THEN
	
	Disable_HV();
	
	IF NOT(DeanStatus.OverCurrentSetpointError) THEN
		DeanStatus.OverCurrentSetpointError := TRUE;
		TraceWithSeverity(Message := 'Current limit exceeded', severity := TcEventSeverity.Error);
	END_IF
	
END_IF

// Check for voltage errors
IF 		DeanConfig.HasVMON
	AND DeanStatus.VMON > DeanConfig.MaxVoltageAbs + DeanConfig.MaxVoltageBuffer THEN
	
	Disable_HV();
	InputPowerOff();
	
	IF NOT(DeanStatus.OverMaxVoltageError) THEN
		DeanStatus.OverMaxVoltageError := TRUE;
		TraceWithSeverity(Message := 'HVPS max output voltage exceeded', severity := TcEventSeverity.Critical);
	END_IF
	
ELSIF 	DeanConfig.HasVMON
	AND DeanConfig.HasVSET
	AND DeanStatus.VMON > (DeanConfig.OverVoltageErrorThreshold * DeanConfig.VSET)
	AND DeanConfig.VSET > 0 THEN
	
	Disable_HV();
	
	IF NOT(DeanStatus.OverVoltageSetpointError) THEN
		DeanStatus.OverVoltageSetpointError := TRUE;
		TraceWithSeverity(Message := 'Voltage setpoint exceeded', severity := TcEventSeverity.Error);
	END_IF
END_IF

DeanStatus.ErrorsAreClear := NOT(	DeanStatus.OverCurrentSetpointError OR
									DeanStatus.OverMaxCurrentError 		OR
									DeanStatus.OverVoltageSetpointError OR
									DeanStatus.OverMaxVoltageError		);
END_METHOD

METHOD ClearErrors : BOOL
VAR_INPUT
END_VAR
DeanStatus.OverVoltageSetpointError 	:= FALSE;
DeanStatus.OverMaxVoltageError		 	:= FALSE;
DeanStatus.OverCurrentSetpointError 	:= FALSE;
DeanStatus.OverMaxCurrentError		 	:= FALSE;

DeanStatus.ErrorsAreClear 					:= TRUE;
END_METHOD

METHOD InjectConfiguration
VAR_INPUT
	PowerSupplyConfiguration : REFERENCE TO ST_PowerSupplyConfiguration;
END_VAR
DeanConfig := PowerSupplyConfiguration;
END_METHOD

METHOD Interpolate : LREAL
VAR_INPUT
	Input		: LREAL;
	Input_min 	: LREAL;
	Input_max 	: LREAL;
	Output_min	: LREAL;
	Output_max	: LREAL;
END_VAR
VAR
	Fraction_along : LREAL;
END_VAR
IF Input_max <> Input_min THEN // avoids division by 0
	Fraction_along := (Input - Input_min) / (Input_max - Input_min);
	Interpolate := (Output_max - Output_min) * Fraction_along + Output_min;
ELSE
	Interpolate := Input_min;
END_IF
END_METHOD

PROPERTY P_PowerSupplyConfiguration : REFERENCE TO ST_PowerSupplyConfiguration
GET
P_PowerSupplyConfiguration REF= DeanConfig;
END_GET
END_PROPERTY

PROPERTY P_PowerSupplyStatus : REFERENCE TO ST_PowerSupplyStatus
GET
P_PowerSupplyStatus REF= DeanStatus;
END_GET
END_PROPERTY

END_FUNCTION_BLOCK

// POUs/FB_HVPS_System
FUNCTION_BLOCK FB_HVPS_System EXTENDS FB_BaseCyclic IMPLEMENTS I_PowerSupplySystem
VAR CONSTANT
	INDEX_MIN		: DINT := 0;
	INDEX_TopPos	: DINT := 0;
	INDEX_TopNeg	: DINT := 1;
	INDEX_BotPos	: DINT := 2;
	INDEX_BotNeg	: DINT := 3;
	INDEX_MAX		: DINT := 3;
END_VAR
VAR
	PowerSupplies	: ARRAY[INDEX_MIN..INDEX_MAX] OF FB_DeanPowerSupply;
	iPowerSupplies	: ARRAY[INDEX_MIN..INDEX_MAX] OF I_PowerSupplyExt;
	iPSConfigs		: ARRAY[INDEX_MIN..INDEX_MAX] OF I_PowerSupplyConfiguration;
	
	LoopIndex		: DINT;
	
	PS_Configs		: ARRAY[INDEX_MIN..INDEX_MAX] OF ST_PowerSupplyConfiguration;
	
	run_tests_trigger : BOOL := FALSE;
	test_results : ARRAY[0..7] OF ARRAY[0..3] OF BOOL;
	
	action_triggers	: ARRAY[0..10] OF BOOL;
END_VAR

// Basic component initialization logic
METHOD PROTECTED _Initialize : BOOL;
// This method is called by CyclicLogic() as required
VAR
	InterimInit : BOOL;
END_VAR
// Initialize children dependencies first
InterimInit := _InitializeChildrenDependencies();
IF NOT InterimInit THEN
	IF BaseConfiguration.LogTraceConfiguration.What.xLogToEventLogger AND NOT BaseStatus.LogTraceStatus.InitChildrenFailureShown THEN
		TraceWithSeverity(Message := Tc2_Standard.CONCAT('_InitializeChildrenDependencies Failed at ', __POUNAME()), Severity := Global.TcEventSeverity.Error);
		BaseStatus.LogTraceStatus.InitChildrenFailureShown := TRUE;
	END_IF
	_Initialize := FALSE;
	RETURN;
END_IF

// Initialize references second
InterimInit := _InitializeReferences();
IF NOT InterimInit THEN
	IF BaseConfiguration.LogTraceConfiguration.What.xLogToEventLogger AND NOT BaseStatus.LogTraceStatus.InitReferencesFailureShown THEN
		TraceWithSeverity(Message := Tc2_Standard.CONCAT('_InitializeReferences Failed at ', __POUNAME()), Severity := Global.TcEventSeverity.Error);
		BaseStatus.LogTraceStatus.InitReferencesFailureShown := TRUE;
	END_IF
	_Initialize := FALSE;
	RETURN;
END_IF

// Set dependency configuration last
InterimInit := _SetDependencyConfiguration();
IF NOT InterimInit THEN
	IF BaseConfiguration.LogTraceConfiguration.What.xLogToEventLogger AND NOT BaseStatus.LogTraceStatus.InitDependencyConfigFailureShown THEN
		TraceWithSeverity(Message := Tc2_Standard.CONCAT('_SetDependencyConfiguration Failed at ', __POUNAME()), Severity := Global.TcEventSeverity.Error);
		BaseStatus.LogTraceStatus.InitDependencyConfigFailureShown := TRUE;
	END_IF
	_Initialize := FALSE;
	RETURN;
END_IF

//splice in 
FOR LoopIndex := LOWER_BOUND(PowerSupplies,1) TO UPPER_BOUND(PowerSupplies,1) BY 1 DO
	IF iPowerSupplies[LoopIndex] <> 0 THEN
		// iPowerSupplies[LoopIndex].InjectConfiguration(PowerSupplyConfiguration := astPSConfig[LoopIndex]); //pick one
		iPSConfigs[LoopIndex].P_PowerSupplyConfiguration	:= PS_Configs[LoopIndex];
	END_IF
END_FOR

// All initialization steps succeeded
_Initialize := TRUE;
END_METHOD

METHOD PROTECTED _InitializeChildrenDependencies : BOOL
//Interface Assignment/Wiring
FOR LoopIndex := LOWER_BOUND(PowerSupplies,1) TO UPPER_BOUND(PowerSupplies,1) BY 1 DO
	PowerSupplies[LoopIndex].Initialize();
END_FOR

_InitializeChildrenDependencies := TRUE;
END_METHOD

METHOD PROTECTED _SetDependencyConfiguration : BOOL
FOR LoopIndex := LOWER_BOUND(PowerSupplies,1) TO UPPER_BOUND(PowerSupplies,1) BY 1 DO
	//PowerSupplies[LoopIndex].P_PowerSupplyConfiguration := 
END_FOR

_SetDependencyConfiguration	:= TRUE;
END_METHOD

METHOD CyclicLogic
VAR
END_VAR
SUPER^.CyclicLogic();

// Run the cyclic logic for each power supply
FOR LoopIndex := LOWER_BOUND(PowerSupplies,1) TO UPPER_BOUND(PowerSupplies,1) BY 1 DO
	PowerSupplies[LoopIndex].CyclicLogic();
END_FOR

// Run tests if requested
IF run_tests_trigger THEN
	test_results := RunTests();
	run_tests_trigger := FALSE;
END_IF	

IF action_triggers[0] THEN
	ClearErrors(INDEX_TopPos);
	ClearErrors(INDEX_TopNeg);
	ClearErrors(INDEX_BotPos);
	ClearErrors(INDEX_BotNeg);
	action_triggers[0] := FALSE;
ELSIF action_triggers[1] THEN
	FullShutDown();
	action_triggers[1] := FALSE;
ELSIF action_triggers[2] THEN
	Disable_HV(INDEX_TopPos);
	Disable_HV(INDEX_TopNeg);
	Disable_HV(INDEX_BotPos);
	Disable_HV(INDEX_BotNeg);
	action_triggers[2] := FALSE;
ELSIF action_triggers[3] THEN
	Enable_HV(INDEX_TopPos);
	Enable_HV(INDEX_TopNeg);
	Enable_HV(INDEX_BotPos);
	Enable_HV(INDEX_BotNeg);
	action_triggers[3] := FALSE;
ELSIF action_triggers[4] THEN
	FullShutDown();
	action_triggers[4] := FALSE;
ELSIF action_triggers[5] THEN
	InputPowerOn(INDEX_TopPos);
	InputPowerOn(INDEX_TopNeg);
	InputPowerOn(INDEX_BotPos);
	InputPowerOn(INDEX_BotNeg);
	action_triggers[5] := FALSE;
ELSIF action_triggers[6] THEN
	InputPowerOff(INDEX_TopPos);
	InputPowerOff(INDEX_TopNeg);
	InputPowerOff(INDEX_BotPos);
	InputPowerOff(INDEX_BotNeg);
	action_triggers[6] := FALSE;
ELSIF action_triggers[7] THEN
	SetCurrent(PowerSupplies[INDEX_TopPos].DeanConfig.MinCurrent, INDEX_TopPos);
	SetCurrent(PowerSupplies[INDEX_TopNeg].DeanConfig.MinCurrent, INDEX_TopNeg);
	SetCurrent(PowerSupplies[INDEX_BotPos].DeanConfig.MinCurrent, INDEX_BotPos);
	SetCurrent(PowerSupplies[INDEX_BotNeg].DeanConfig.MinCurrent, INDEX_BotNeg);
	action_triggers[7] := FALSE;
ELSIF action_triggers[8] THEN
	SetCurrent(PowerSupplies[INDEX_TopPos].DeanConfig.MaxCurrent, INDEX_TopPos);
	SetCurrent(PowerSupplies[INDEX_TopNeg].DeanConfig.MaxCurrent, INDEX_TopNeg);
	SetCurrent(PowerSupplies[INDEX_BotPos].DeanConfig.MaxCurrent, INDEX_BotPos);
	SetCurrent(PowerSupplies[INDEX_BotNeg].DeanConfig.MaxCurrent, INDEX_BotNeg);
	action_triggers[8] := FALSE;
ELSIF action_triggers[9] THEN
	SetVoltage(PowerSupplies[INDEX_TopPos].DeanConfig.MinVoltage, INDEX_TopPos);
	SetVoltage(PowerSupplies[INDEX_TopNeg].DeanConfig.MinVoltage, INDEX_TopNeg);
	SetVoltage(PowerSupplies[INDEX_BotPos].DeanConfig.MinVoltage, INDEX_BotPos);
	SetVoltage(PowerSupplies[INDEX_BotNeg].DeanConfig.MinVoltage, INDEX_BotNeg);
	action_triggers[9] := FALSE;
ELSIF action_triggers[10] THEN
	SetVoltage(PowerSupplies[INDEX_TopPos].DeanConfig.MaxVoltageAbs, INDEX_TopPos);
	SetVoltage(PowerSupplies[INDEX_TopNeg].DeanConfig.MaxVoltageAbs, INDEX_TopNeg);
	SetVoltage(PowerSupplies[INDEX_BotPos].DeanConfig.MaxVoltageAbs, INDEX_BotPos);
	SetVoltage(PowerSupplies[INDEX_BotNeg].DeanConfig.MaxVoltageAbs, INDEX_BotNeg);
	action_triggers[10] := FALSE;
END_IF
END_METHOD

//FB_Init is always available implicitly and it is used primarily for initialization.
//The return value is not evaluated. For a specific influence, you can also declare the
//methods explicitly and provide additional code there with the standard initialization
//code. You can evaluate the return value.
METHOD FB_Init: BOOL
VAR_INPUT
    bInitRetains: BOOL; // TRUE: the retain variables are initialized (reset warm / reset cold)
    bInCopyCode: BOOL;  // TRUE: the instance will be copied to the copy code afterward (online change)   
END_VAR
//Interface Assignment/Wiring
FOR LoopIndex := LOWER_BOUND(PowerSupplies,1) TO UPPER_BOUND(PowerSupplies,1) BY 1 DO
	iPowerSupplies[LoopIndex]	:= PowerSupplies[LoopIndex];
	iPSConfigs[LoopIndex]		:= PowerSupplies[LoopIndex];
END_FOR

// Populating DeanConfig
// Assign everything that is the same for all four supplies
FOR LoopIndex := LOWER_BOUND(PowerSupplies,1) TO UPPER_BOUND(PowerSupplies,1) BY 1 DO

	PS_Configs[LoopIndex].MinVoltage 		:= 0;
	PS_Configs[LoopIndex].MaxVoltageAbs 	:= 6000;
	PS_Configs[LoopIndex].MinCurrent 		:= 0;
	PS_Configs[LoopIndex].MaxCurrent	 	:= 1; // This is much higher than we should need
	
	PS_Configs[LoopIndex].NeedsVREF 		:= FALSE;
	PS_Configs[LoopIndex].HasVMON		 	:= FALSE;
	PS_Configs[LoopIndex].HasVSET		 	:= TRUE;
	PS_Configs[LoopIndex].HasISET		 	:= TRUE;
	PS_Configs[LoopIndex].HasIMON		 	:= TRUE;     

	PS_Configs[LoopIndex].plc_min_VSET  	:= 0;	 
	PS_Configs[LoopIndex].plc_max_VSET 		:= 32767;                            
	PS_Configs[LoopIndex].plc_min_ISET  := LREAL_TO_INT(FLOOR(PS_Configs[LoopIndex].MinCurrent / 3.3 * 32767)); 
	PS_Configs[LoopIndex].plc_max_ISET  := LREAL_TO_INT(FLOOR(PS_Configs[LoopIndex].MaxCurrent / 3.3 * 32767));
	PS_Configs[LoopIndex].plc_min_IMON  := LREAL_TO_INT(FLOOR(PS_Configs[LoopIndex].MinCurrent / 3.3 * 10.0 / 10.73 * 32767));  // 0	 
	PS_Configs[LoopIndex].plc_max_IMON  := LREAL_TO_INT(FLOOR(PS_Configs[LoopIndex].MaxCurrent / 3.3 * 10.0 / 10.73 * 32767));

	PS_Configs[LoopIndex].OverCurrentErrorThreshold := 1.10; // default 1.05
END_FOR

// Assign things that are different between supplies
PS_Configs[INDEX_TopPos].IsPositive 	:= 	TRUE	;
PS_Configs[INDEX_TopNeg].IsPositive 	:= 	FALSE	;
PS_Configs[INDEX_BotPos].IsPositive 	:= 	TRUE 	;
PS_Configs[INDEX_BotNeg].IsPositive 	:= 	FALSE	;

PS_Configs[INDEX_TopPos].VSET_needs_ramp 	:= 	FALSE	;
PS_Configs[INDEX_TopNeg].VSET_needs_ramp 	:= 	FALSE	;
PS_Configs[INDEX_BotPos].VSET_needs_ramp 	:= 	TRUE 	;
PS_Configs[INDEX_BotNeg].VSET_needs_ramp 	:= 	TRUE	;

PS_Configs[INDEX_BotPos].Ramp_increment := 20;
PS_Configs[INDEX_BotNeg].Ramp_increment := 20;

// V out * (V mon / V out) scaling ÷ V terminal range * dimensionless terminal range                                 
// 	PS_Configs[LoopIndex].plc_min_VMON  := LREAL_TO_INT(PS_Configs[LoopIndex].MinVoltage * 0.01 / 64.32 * 32767); 
// 	PS_Configs[LoopIndex].plc_max_VMON  := LREAL_TO_INT(PS_Configs[LoopIndex].MaxVoltageAbs * 0.01 / 64.32 * 32767);  

// PS_Configs[INDEX_TopPos].plc_min_ISET  := 0;	 
// PS_Configs[INDEX_TopPos].plc_max_ISET  := LREAL_TO_INT(FLOOR(32767 * PS_Configs[INDEX_TopPos].VREF / 10.00));
// PS_Configs[INDEX_TopNeg].plc_min_ISET  := 0;	 
// PS_Configs[INDEX_TopNeg].plc_max_ISET  := LREAL_TO_INT(FLOOR(32767 * PS_Configs[INDEX_TopPos].VREF / 10.00));

// mA output * (V/mA) scaling ÷ V terminal range * dimensionless terminal range
// PS_Configs[INDEX_TopPos].plc_min_IMON  := LREAL_TO_INT(FLOOR(PS_Configs[INDEX_TopPos].MinCurrent * (1.0/6.2) / 10.73 * 32767));  // 0
// PS_Configs[INDEX_TopPos].plc_max_IMON  := LREAL_TO_INT(FLOOR(PS_Configs[INDEX_TopPos].MaxCurrent * (1.0/6.2) / 10.73 * 32767));
// PS_Configs[INDEX_TopNeg].plc_min_IMON  := LREAL_TO_INT(FLOOR(PS_Configs[INDEX_TopNeg].MinCurrent * (1.0/6.2) / 10.73 * 32767));  // 0
// PS_Configs[INDEX_TopNeg].plc_max_IMON  := LREAL_TO_INT(FLOOR(PS_Configs[INDEX_TopNeg].MaxCurrent * (1.0/6.2) / 10.73 * 32767)); 

// Temporary fixes to protect the broken half of one supply                                                                                     
// PS_Configs[INDEX_TopPos].MaxVoltageAbs := 4800; 
// PS_Configs[INDEX_TopPos].plc_max_VSET  := LREAL_TO_INT(FLOOR(32767 * (4800.0/6000.0) * PS_Configs[INDEX_TopPos].VREF / 10.00));
END_METHOD

PROPERTY P_supply_status : ARRAY[INDEX_MIN..INDEX_MAX] OF ST_PowerSupplyStatus
GET
FOR LoopIndex := LOWER_BOUND(PowerSupplies,1) TO UPPER_BOUND(PowerSupplies,1) BY 1 DO
	P_supply_status[LoopIndex] := PowerSupplies[LoopIndex].DeanStatus;
END_FOR
END_GET
END_PROPERTY

METHOD RunTests : ARRAY[0..7] OF ARRAY[0..3] OF BOOL
VAR
	Result_Enable_HV		: ARRAY[0..3] OF BOOL;
	Result_Disable_HV		: ARRAY[0..3] OF BOOL;
	Result_InputPowerOn		: ARRAY[0..3] OF BOOL;
	Result_InputPowerOff	: ARRAY[0..3] OF BOOL;
	Result_GetVoltage		: ARRAY[0..3] OF BOOL;
	Result_GetCurrent		: ARRAY[0..3] OF BOOL;
	Result_SetVoltage		: ARRAY[0..3] OF BOOL;
	Result_SetCurrent		: ARRAY[0..3] OF BOOL;
	
	summary_table : ARRAY[0..7] OF POINTER TO ARRAY[0..3] OF BOOL := [ 	ADR(Result_Enable_HV	),
		                                                    			ADR(Result_Disable_HV	),
		                                                    			ADR(Result_InputPowerOn	),
		                                                    			ADR(Result_InputPowerOff),
		                                                    			ADR(Result_GetVoltage	),
		                                                    			ADR(Result_GetCurrent	),
		                                                    			ADR(Result_SetVoltage	),
		                                                    			ADR(Result_SetCurrent	)];	
	loop_index : DINT;
	
	RealConfig : ST_PowerSupplyConfiguration;
	RealStatus : ST_PowerSupplyStatus;
END_VAR
 FOR loop_index := LOWER_BOUND(PowerSupplies,1) TO UPPER_BOUND(PowerSupplies,1) BY 1 DO
	// Store the current state
	RealConfig := PowerSupplies[loop_index].DeanConfig;
	RealStatus := PowerSupplies[loop_index].DeanStatus;

	// Run tests (may change state)
	Result_Enable_HV	[loop_index] 	:= PowerSupplies[loop_index].Test_Enable_HV();
	Result_Disable_HV	[loop_index] 	:= PowerSupplies[loop_index].Test_Disable_HV();
	Result_InputPowerOn	[loop_index] 	:= PowerSupplies[loop_index].Test_InputPowerOn();
	Result_InputPowerOff[loop_index] 	:= PowerSupplies[loop_index].Test_InputPowerOff();
	Result_GetVoltage	[loop_index] 	:= PowerSupplies[loop_index].Test_GetVoltage();
	Result_GetCurrent	[loop_index] 	:= PowerSupplies[loop_index].Test_GetCurrent();
	Result_SetVoltage	[loop_index] 	:= PowerSupplies[loop_index].Test_SetVoltage();
	Result_SetCurrent	[loop_index] 	:= PowerSupplies[loop_index].Test_SetCurrent();
	
	// Restore the original state
	PowerSupplies[loop_index].DeanConfig := RealConfig;
	PowerSupplies[loop_index].DeanStatus := RealStatus;
END_FOR

FOR loop_index := 0 TO 7 BY 1 DO
	RunTests[loop_index] := summary_table[loop_index]^;
END_FOR
END_METHOD

(*Acknowledge and reset over-voltage and over-current errors*)
METHOD ClearErrors : BOOL
VAR_INPUT
	Index : DINT;
END_VAR
PowerSupplies[Index].DeanConfig.ClearErrors := TRUE;
END_METHOD

(* Shut off the output voltage of a supply*)
METHOD Disable_HV
VAR_INPUT
	Index : DINT;
END_VAR
PowerSupplies[Index].DeanConfig.ENABLED := FALSE;
END_METHOD

{warning 'Add method implementation '}
(* Turn on the output voltage of a supply*)
METHOD Enable_HV
VAR_INPUT
	Index : DINT;
END_VAR
PowerSupplies[Index].DeanConfig.ENABLED := TRUE;
END_METHOD

METHOD FullShutDown : BOOL
Disable_HV(0);
Disable_HV(1);
Disable_HV(2);
Disable_HV(3);

InputPowerOff(0);
InputPowerOff(1);
InputPowerOff(2);
InputPowerOff(3);
END_METHOD

{warning 'Add method implementation '}
(* Turn off power to a supply*)
METHOD InputPowerOff
VAR_INPUT
	Index : DINT;
END_VAR
PowerSupplies[Index].DeanConfig.POWERED := FALSE;
END_METHOD

{warning 'Add method implementation '}
(* Turn on power to a supply*)
METHOD InputPowerOn
VAR_INPUT
	Index : DINT;
END_VAR
PowerSupplies[Index].DeanConfig.POWERED := TRUE;
END_METHOD

{warning 'Add method implementation '}
(* Send the the desired or maximum current setpoint (in mA) to a supply*)
METHOD SetCurrent
VAR_INPUT
	(* mA*)
	setpoint	: LREAL;
	Index : DINT;
END_VAR
PowerSupplies[Index].DeanConfig.ISET := setpoint;
END_METHOD

{warning 'Add method implementation '}
(* Send the the voltage setpoint (V) to a supply*)
METHOD SetVoltage
VAR_INPUT
	(* V*)
	setpoint	: LREAL;
	Index : DINT;
END_VAR
PowerSupplies[Index].DeanConfig.VSET := setpoint;
END_METHOD

END_FUNCTION_BLOCK

// POUs/MAIN
PROGRAM MAIN
VAR
	HVPS 			: FB_HVPS_System;				// This instantiates 4 supplies
	iHVPS			: I_PowerSupplySystem := HVPS;
	
	// top_pos_index	: DINT := 0;
	// top_neg_index	: DINT := 0;
	// bot_pos_index	: DINT := 0;
	// bot_neg_index	: DINT := 0;
END_VAR

HVPS.CyclicLogic(); // This actually runs the supplies

// iHVPS is an interface that has all the methods you should need to control the supplies. Example:
// iHVPS.SetVoltage(top_pos_index, 3000);
// iHVPS does not allow configuration changes beyond those related to control.

// HVPS.P_supply_status is a read-only property that you can use to access current status for the supplies. Example:
// ReadyToCut 	:= 	HVPS.P_supply_status[bot_neg_index].POWERED AND (HVPS.P_supply_status[bot_neg_index].VSET = 6000);

// I think if you like you can also just map these variables directly in the HMI:
// Go to the ADS variables and look for, for example, 'HVPS.P_supply_status[top_pos_index].IMON' and then map it (just remember these are read-only)

END_PROGRAM
